// TIA Portal V16 export
// export: Created 2023-08-28T09:37:48.1818354Z, ExportSetting WithDefaults, DisplayName Totally Integrated Automation Portal, DisplayVersion V16 Update 6, DisplayName TIA Portal Version Control Interface, DisplayVersion V16 Update 2, DisplayName TIA Portal Openness, DisplayVersion V16 Update 6, DisplayName STEP 7 Professional, DisplayVersion V16 Update 6, DisplayName STEP 7 Safety, DisplayVersion V16, DisplayName WinCC Advanced, DisplayVersion V16 Update 6
DATA_BLOCK "dbControl of   Inverters_DB"   // DB49
AUTHOR : rtecmer
VERSION : 0.1
// stored: AutoNumber true, DBAccessibleFromOPCUA true, InstanceOfName 06_M_Inverte control, InstanceOfType FB
"06_M_Inverte control"
   // VAR_INPUT
   //    IsModeAut : Bool;
   //    AlwaysTRUE : Bool;
   //    Set_HWork_P1 : Bool;
   //    Set_HWork_P2 : Bool;
   //    Set_HWork_P3 : Bool;
   //    Set_HWork_P4 : Bool;
   //    setPID_Pomp : Bool;
   //    Is_loading_K3 : Bool;
   //    IsRunInverter_P4 : Bool;
   //    IsRunInverter_P3 : Bool;
   //    IsRunInverter_P2 : Bool;
   //    IsRunInverter_P1 : Bool;
   //    Bit_Aut_P1 : Bool;
   //    Bit_Aut_P2 : Bool;
   //    Bit_Aut_P3 : Bool;
   //    Bit_Aut_P4 : Bool;
   //    IsRunNetwork_P1 : Bool;
   //    IsRunNetwork_P2 : Bool;
   //    IsRunNetwork_P3 : Bool;
   //    IsRunNetwork_P4 : Bool;
   // END_VAR
   // VAR_OUTPUT
   //    CMD_start_stop_inverter : Bool;
   // END_VAR
   // VAR
   //    Res_upHz : Bool;
   // END_VAR
BEGIN
END_DATA_BLOCK
